PROGRAM GearingFlyingSaw
VAR
	iGearMode				: UDINT;
	
	GearInDyn				: MC_GearInDyn;
	bGearInDynActive		: BOOL;
	lrGearRatio				: LREAL :=1.0;
	
	bFlyingSawActive		: BOOL;
	FlyingSaw				: MC_GearInPos;
	SyncMode           		: ST_SyncMode;

	GearOut					: MC_GearOut;
	
	// Master Trigger and Master / Slave sync positions
	lrMasterTrigPos			: LREAL :=360;
	lrMasterSyncPos			: LREAL :=720;
	lrSlaveSyncPos			: LREAL :=720;
	

END_VAR

IF iGearMode=1 THEN
	bGearInDynActive:=TRUE;
END_IF

(* trigger Flying Saw -- can be any boolean condition or digital input *)
IF bMvMstr AND iGearMode=2 AND axs_Mstr.NcToPlc.ActPos>lrMasterTrigPos THEN
	bFlyingSawActive:=TRUE;
	bGearInDynActive:=FALSE;	
END_IF

IF iGearMode=0 THEN
	bGearInDynActive:=FALSE;	
	bFlyingSawActive:=FALSE;
END_IF

IF NOT(mv_MasterAbs.Busy) AND NOT(mv_MasterRel.Busy) THEN
	bFlyingSawActive:=FALSE;
END_IF

GearFS_FBs();

ACTION GearFS_FBs:
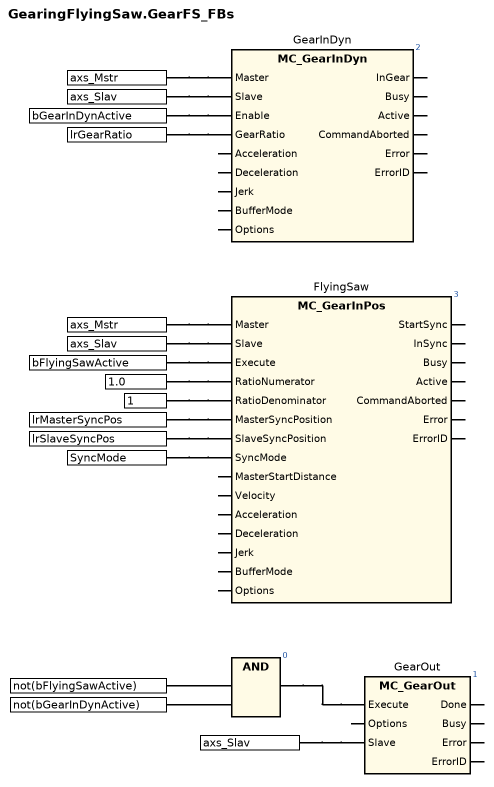
GearOut(Execute := (not(bFlyingSawActive)) AND (not(bGearInDynActive)), Slave := axs_Slav); // MC_GearOut
GearInDyn(Master := axs_Mstr, Slave := axs_Slav, Enable := bGearInDynActive, GearRatio := lrGearRatio); // MC_GearInDyn
FlyingSaw(
    Master := axs_Mstr,
    Slave := axs_Slav,
    Execute := bFlyingSawActive,
    RatioNumerator := 1.0,
    RatioDenominator := 1,
    MasterSyncPosition := lrMasterSyncPos,
    SlaveSyncPosition := lrSlaveSyncPos,
    SyncMode := SyncMode); // MC_GearInPos
END_ACTION

END_PROGRAM

(* stored: Version 1.1.0.1, ProductVersion 3.1.4024.11
   POU GearingFlyingSaw: Id {a8f82dba-ca4e-4533-a5e8-b294a7bec4f9}, SpecialFunc None
   Action GearFS_FBs: Id {b838319d-e230-4149-ae0f-209bc9e1126a} *)
